(* IEC 61131-3 sources: Std_PalletMover/Class/Curtis_Base, 1 file *)

(* ---- Curtis_Base.st ---- *)
//#Define cNoNmtIfOk
#Define cCommTo                   1000    // 1000
#Define cHeartBeat                150     // 1000 Every 1 Sec.
#define COMM_TIMEOUT              1000    // ms before timeout
#define PDO1_SEND_INTERVAL        40      // 100 ms
#define TIMEOUTDELAY              15000    // Delay before checking for a communication timeout.
#define REFERENCETIMEOUT          30 SEC  //
#define FUSE_BAD_TIME             4 SEC
#define MAX_TIME_DRIVE_MODE_REQ   150 //ms

(*!
<Class
	Name               = "Curtis_Base"
	Revision           = "0.0"
	RealtimeTask       = "false"
	CyclicTask         = "false"
	DefCyclictime      = "5 ms"
	BackgroundTask     = "false"
	Sigmatek           = "false"
	OSInterface        = "false"
	HighPriority       = "false"
	Automatic          = "false"
	UpdateMode         = "Prescan"
	IconPath           = ".\Class\Curtis_1232E_FR\curtis.ico"
	SharedCommandTable = "true"
	Objectsize         = "(510,300)"
	Comment            = "CAN Message for Curtis Drives">
	<Channels>
		<Server Name="Active" Visualized="true" Initialize="false" WriteProtected="true" Retentive="false"/>
		<Server Name="AI_BrakePot" Visualized="true" Initialize="false" WriteProtected="true" Retentive="false"/>
		<Server Name="AI_ThrottlePot" Visualized="true" Initialize="false" WriteProtected="true" Retentive="false"/>
		<Server Name="AutoAccelTime" Visualized="true" Initialize="true" DefValue="100" WriteProtected="false" Retentive="SRam" Comment="0,1 second acceleration time"/>
		<Server Name="AutoAct" Visualized="true" Initialize="false" WriteProtected="true" Retentive="false"/>
		<Server Name="AutoDecelTime" Visualized="true" Initialize="true" DefValue="10" WriteProtected="false" Retentive="SRam" Comment="0,1 second acceleration time"/>
		<Server Name="AutomaticSetpoint" Visualized="true" Initialize="false" WriteProtected="false" Retentive="false"/>
		<Server Name="AutoSetp" Visualized="true" Initialize="false" WriteProtected="true" Retentive="false"/>
		<Server Name="BDI" Visualized="true" Initialize="false" WriteProtected="true" Retentive="false"/>
		<Server Name="BrakePotSigned" Visualized="true" Initialize="true" WriteProtected="false" Retentive="File"/>
		<Server Name="Capacitor_Voltage" Visualized="true" Initialize="false" WriteProtected="true" Retentive="false"/>
		<Server Name="ClassSvr" Visualized="false" Initialize="false" WriteProtected="true" Retentive="false"/>
		<Server Name="CommunicationOk" Visualized="true" Initialize="false" WriteProtected="true" Retentive="false"/>
		<Server Name="DriveMode" Visualized="true" Initialize="false" WriteProtected="true" Retentive="false"/>
		<Server Name="DriveModeRequest" Visualized="true" Initialize="false" WriteProtected="false" Retentive="false"/>
		<Server Name="EmStopOk" Visualized="true" Initialize="false" WriteProtected="true" Retentive="false"/>
		<Server Name="Enabled" Visualized="true" Initialize="true" DefValue="1" WriteProtected="false" Retentive="File"/>
		<Server Name="I_DigitalOut6" Visualized="true" Initialize="false" WriteProtected="true" Retentive="false" Comment="Sw_14"/>
		<Server Name="I_DigitalOut7" Visualized="true" Initialize="false" WriteProtected="true" Retentive="false" Comment="Sw_15"/>
		<Server Name="I_Driver1" Visualized="true" Initialize="false" WriteProtected="true" Retentive="false" Comment="Sw_9&#13;&#10;Auger_1 - bI_SP_HighLow"/>
		<Server Name="I_Driver2" Visualized="true" Initialize="false" WriteProtected="true" Retentive="false" Comment="Sw_10&#13;&#10;Auger_1 - bI_AugerOnOff"/>
		<Server Name="I_Driver3" Visualized="true" Initialize="false" WriteProtected="true" Retentive="false" Comment="Sw_11&#13;&#10;Auger_1 - bSP_HighLow"/>
		<Server Name="I_Driver4" Visualized="true" Initialize="false" WriteProtected="true" Retentive="false" Comment="Sw_12&#13;&#10;Auger_1 - bAugerOnOff"/>
		<Server Name="I_PropDriver" Visualized="true" Initialize="false" WriteProtected="true" Retentive="false" Comment="Sw_13&#13;&#10;Pin 2"/>
		<Server Name="I_Switch1" Visualized="true" Initialize="false" WriteProtected="true" Retentive="false" Comment="Pin 24 - Switch 1"/>
		<Server Name="I_Switch16" Visualized="true" Initialize="false" WriteProtected="true" Retentive="false" Comment="Pin 14 - Switch 16"/>
		<Server Name="I_Switch2" Visualized="true" Initialize="false" WriteProtected="true" Retentive="false" Comment="Pin 8 - Switch 2"/>
		<Server Name="I_Switch3" Visualized="true" Initialize="false" WriteProtected="true" Retentive="false" Comment="Pin 9 - Switch 3"/>
		<Server Name="I_Switch4" Visualized="true" Initialize="false" WriteProtected="true" Retentive="false" Comment="Pin 10 - Switch 4"/>
		<Server Name="I_Switch5" Visualized="true" Initialize="false" WriteProtected="true" Retentive="false" Comment="Pin 11 - Switch 5"/>
		<Server Name="I_Switch6" Visualized="true" Initialize="false" WriteProtected="true" Retentive="false" Comment="Pin 12 - Switch 6"/>
		<Server Name="I_Switch7" Visualized="true" Initialize="false" WriteProtected="true" Retentive="false" Comment="Pin 22 - Switch 7"/>
		<Server Name="I_Switch8" Visualized="true" Initialize="false" WriteProtected="true" Retentive="false" Comment="Pin 33 - Switch 8"/>
		<Server Name="InterlockExternal1" Visualized="true" Initialize="false" WriteProtected="true" Retentive="false"/>
		<Server Name="InterlockExternal2" Visualized="true" Initialize="false" WriteProtected="true" Retentive="false"/>
		<Server Name="InterlockFeedback" Visualized="true" Initialize="false" WriteProtected="true" Retentive="false"/>
		<Server Name="MotorCurrent" Visualized="true" Initialize="false" WriteProtected="true" Retentive="false"/>
		<Server Name="MotorRPM" Visualized="true" Initialize="false" WriteProtected="true" Retentive="false" Comment="Speed of Motor"/>
		<Server Name="MotorTemperature" Visualized="true" Initialize="false" WriteProtected="true" Retentive="false"/>
		<Server Name="QD_DigitalOut6" Visualized="true" Initialize="false" WriteProtected="false" Retentive="false" Comment="Auger_1 - Horn"/>
		<Server Name="QD_DigitalOut7" Visualized="true" Initialize="false" WriteProtected="false" Retentive="false" Comment="Auger_1 - bDrive_OnOff"/>
		<Server Name="QD_Driver1" Visualized="true" Initialize="false" WriteProtected="false" Retentive="false" Comment="Auger_1 - Pin 6 - bQ_Actu_L_In"/>
		<Server Name="QD_Driver2" Visualized="true" Initialize="false" WriteProtected="false" Retentive="false" Comment="Auger_1 - Pin 5 - bQ_Actu_L_Out"/>
		<Server Name="QD_Driver3" Visualized="true" Initialize="false" WriteProtected="false" Retentive="false" Comment="Auger_1 - Pin 4 - bQ_Actu_R_In"/>
		<Server Name="QD_Driver4" Visualized="true" Initialize="false" WriteProtected="false" Retentive="false" Comment="Auger_1 - Pin 3 - bQ_Actu_R_Out"/>
		<Server Name="QD_PropDriver" Visualized="true" Initialize="false" WriteProtected="false" Retentive="false"/>
		<Server Name="Referenced" Visualized="true" Initialize="false" WriteProtected="true" Retentive="false"/>
		<Server Name="ThrottlePotSigned" Visualized="true" Initialize="true" WriteProtected="false" Retentive="File"/>
		<Client Name="_CanOpenBaseRiwo" Required="true" Internal="true"/>
		<Client Name="AlarmStartId" Required="true" Internal="false"/>
		<Client Name="NodeId" Required="true" Internal="false"/>
		<Client Name="objDriver" Required="false" Internal="false"/>
	</Channels>
	<Separators>
		<Servers>
			<SepChn Position="34"/>
			<SepChn Position="38"/>
		</Servers>
	</Separators>
	<RevDoku>
		<Owner Company="RIWO Engineering BV" Author="P vd Voort"/>
		<Dokumentation Revision="0.0" Date="2022-08-29" Author="P vd Voort" Company="RIWO Engineering BV" Description="First Build Up"/>
	</RevDoku>
	<Network Name="Curtis_Base">
		<!-- List of Components in this network -->
		<Components>
			<Object
				Name       = "_CanOpenBaseRiwo"
				Class      = "CanOpenBaseRiwo"
				Position   = "(390,240)"
				Visualized = "true"
				CyclicTime = "1 ms">
				<Channels>
					<Server Name="Server0"/>
					<Client Name="cNode" Value="1"/>
					<Client Name="ConfigData"/>
					<Client Name="Driver"/>
				</Channels>
			</Object>
		</Components>
		<Comments>
		</Comments>
		<!-- List of Connections in this network -->
		<Connections>
			<Connection Source="this._CanOpenBaseRiwo" Destination="_CanOpenBaseRiwo.Server0"/>
			<Connection Source="_CanOpenBaseRiwo.Driver" Destination="this.objDriver" Vertices="(390,330),(38,330),"/>
			<Connection Source="_CanOpenBaseRiwo.cNode" Destination="this.NodeId" Vertices="(390,390),(38,270),"/>
		</Connections>
		<!-- Headerfiles -->
		<Options>
		</Options>
	</Network>
</Class>
*)
Curtis_Base : CLASS
	TYPE
#pragma pack(push, 1)
	  CurtisMessageConfig : STRUCT
	    Byte0 : BSINT
	    [
	      1 Q1,
	      2 Q1not,
	      3 Q2,
	      4 Q2not,
	      5 Bit4,
	      6 Bit5,
	      7 Bit6,
	      8 Bit7,
	    ];
	    Byte1 : BSINT
	    [
	      1 InputState_A,
	      2 InputState_B,
	      3 InputState_C,
	      4 InputState_D,
	      5 Bit4,
	      6 Bit5,
	      7 Bit6,
	      8 InputState_StandBy,
	    ];
	    Byte2 : BSINT
	    [
	      1 Bit0_SwFldQ1,
	      2 Bit1_SwFldQ1,
	      3 Bit2_SwFldQ1,
	      4 Bit3_SwFldQ1,
	      5 Bit4_SwFldQ1,
	      6 Bit5,
	      7 Bit6,
	      8 Bit7,
	    ];
	    Byte3 : BSINT
	    [
	      1 Bit0_SwFldQ2,
	      2 Bit1_SwFldQ2,
	      3 Bit2_SwFldQ2,
	      4 Bit3_SwFldQ2,
	      5 Bit4_SwFldQ2,
	      6 Bit5,
	      7 Bit6,
	      8 Bit7,
	    ];
	    Byte4 : BSINT
	    [
	      1 Bit0_DeviceStatus,
	      2 Bit1_DeviceStatus,
	      3 Bit2_DeviceStatus,
	      4 Bit3_DeviceStatus,
	      5 Bit4,
	      6 Bit5,
	      7 Bit6,
	      8 Bit7,
	    ];
	    Byte5 : SINT;
	    Byte6and7 : INT;
	  END_STRUCT;
#pragma pack(pop)
	  CurtisSendConfig : BSINT
	  [
	    1 VirtInp_A,
	    2 VirtInp_B,
	    3 VirtInp_C,
	    4 VirtInp_D,
	    5 Bit4,
	    6 Bit5,
	    7 Bit6,
	    8 VirtInp_Standby,
	  ];
	  eCurtisAlarms :
	  (
	    ca_MainContactor_Welded:=1,
	    ca_MainContactor_NotClosed:=2,
	    ca_PotLow:=3,
	    ca_ThrottleLow:=4,
	    ca_ThrottleHigh:=5,
	    ca_Pot2Low:=6,
	    ca_Pot2High:=7,
	    ca_EepromFail:=8,
	    ca_SequenceFault:=9,
	    ca_UnderVoltage:=10,
	    ca_OverVoltage:=11,
	    ca_UnderVoltage_CutBack:=12,
	    ca_OverVoltage_CutBack:=13,
	    ca_FuseBad:=14,
	    ca_ControllerTemp_CutBack:=15,
	    ca_Controller_UnderTemp:=16,
	    ca_Controller_OverTemp:=17,
	    ca_Coil1_Short:=18,
	    ca_Coil2_Short:=19,
	    ca_Coil3_Short:=20,
	    ca_Coil4_Short:=21,
	    ca_PD_Short:=22,
	    ca_Main_Short:=23,
	    ca_EmBrake_Short:=24,
	    ca_PreCharge_Failed:=25,
	    ca_Digital6_OverCurrent:=26,
	    ca_Digital7_OverCurrent:=27,
	    ca_Controller_OverCurrent:=28,
	    ca_CurrentSensor_Fault:=29,
	    ca_MotorTemp_CutBack:=30,
	    ca_ParameterChange_Fault:=31,
	    ca_Motor_Open:=32,
	    ca_ExtSupply_OutofRange:=33,
	    ca_MotorTemp_SensorFault:=34,
	    ca_VC1_RunTime:=35,
	    ca_5vSupply_Failure:=36,
	    ca_OSGeneral:=37,
	    ca_PDO_Timeout:=38,
	    ca_Encoder_Fault:=39,
	    ca_StallDetected:=40,
	    ca_Com_Timeout:=41,
	    ca_NotRef:=42,
	    ca_RevHpd:=43,
	    ca_NotEnabled:=44,
	    ca_MotorType_Fault:=45,
	    ca_SuperVision:=46,
	    ca_MotorCharacter:=47,
	    ca_PumpHardware:=48,
	    ca_NotDefined_1:=49,
	    ca_VCL_Mismatch:=50,
	    ca_EmBrake_Failed:=51,
	    ca_Encoder_Lose:=52,
	    ca_Rev_Timeout:=53,
	    ca_Dual_Fault:=54,
	    ca_TractionController_Fault:=55,
	    ca_Illegal_ModelNumber:=56,
	    ca_PumpOverCurrent:=57,
	    ca_PumpBdi:=58,
	    ca_PumpHpd:=59,
	    ca_DualMotor_Par_MisMatch:=60,
	    ca_NotDefined_2:=61,
	    ca_NotDefined_3:=62,
	    ca_NotDefined_4:=63,
	    ca_EncoderPulse:=64
	  )$UDINT;
	  eCurtisDriveMode :  //! <Type Public="true" Name="eCurtisDriveMode"/>
	  (
	    cdm_Idle,
	    cdm_TimeOut,
	    cdm_EmergencyStop,
	    cdm_Referencing,
	    cdm_Manual,
	    cdm_Auto,
	    cdm_DriveReset,
	    cdm_ExtInterlockReset
	  )$UDINT;
	  eCurtisDriveModeRequest :  //! <Type Public="true" Name="eCurtisDriveModeRequest"/>
	  (
	    cdmr_NoReq:=4294967295,
	    cdmr_Idle,
	    cdmr_Reference,
	    cdmr_Manual:=2,
	    cdmr_Automatic:=3,
	    cdmr_ResetDrive:=4,
	    cdmr_ResetExtInterlock:=5
	  )$DINT;
#pragma pack(push, 1)
	  Errors : STRUCT
	    Error1 : DINT;
	    Error2 : DINT;
	    Error3 : DINT;
	    Error4 : DINT;
	    Error5 : DINT;
	    Error6 : DINT;
	    Error7 : DINT;
	    NumberOfErrors : DINT;
	  END_STRUCT;
#pragma pack(pop)
	  FuncComm :
	  (
	    _StandBy,
	    _Read,
	    _Write,
	    _Busy
	  )$UDINT;
#pragma pack(push, 1)
	  PdoSplit : STRUCT
	    Val1 : HSINT;
	    Val2 : HSINT;
	    Val3 : HSINT;
	    Val4 : HSINT;
	    Val5 : HSINT;
	    Val6 : HSINT;
	    Val7 : HSINT;
	    Val8 : HSINT;
	  END_STRUCT;
#pragma pack(pop)
	END_TYPE
  //Servers:
	ClassSvr 	: SvrChCmd_DINT;
	Active 	: SvrCh_DINT;
	CommunicationOk 	: SvrCh_DINT;
	DriveMode 	: SvrCh_eCurtisDriveMode_PTofCls_Curtis_Base;
	EmStopOk 	: SvrCh_DINT;
	Referenced 	: SvrCh_DINT;
	InterlockFeedback 	: SvrCh_DINT;
	InterlockExternal1 	: SvrCh_DINT;
	InterlockExternal2 	: SvrCh_DINT;
	AutoAct 	: SvrCh_DINT;
	AutoSetp 	: SvrCh_DINT;
	MotorCurrent 	: SvrCh_DINT;
	BDI 	: SvrCh_DINT;
	Capacitor_Voltage 	: SvrCh_DINT;
	MotorTemperature 	: SvrCh_DINT;
	AI_ThrottlePot 	: SvrCh_DINT;
	AI_BrakePot 	: SvrCh_DINT;
	I_Switch1 	: SvrCh_DINT;
	I_Switch2 	: SvrCh_DINT;
	I_Switch3 	: SvrCh_DINT;
	I_Switch4 	: SvrCh_DINT;
	I_Switch5 	: SvrCh_DINT;
	I_Switch6 	: SvrCh_DINT;
	I_Switch7 	: SvrCh_DINT;
	I_Switch8 	: SvrCh_DINT;
	I_Driver1 	: SvrCh_DINT;
	I_Driver2 	: SvrCh_DINT;
	I_Driver3 	: SvrCh_DINT;
	I_Driver4 	: SvrCh_DINT;
	I_PropDriver 	: SvrCh_DINT;
	I_DigitalOut6 	: SvrCh_DINT;
	I_DigitalOut7 	: SvrCh_DINT;
	I_Switch16 	: SvrCh_DINT;
	MotorRPM 	: SvrCh_DINT;
	Enabled 	: SvrCh_DINT;
	ThrottlePotSigned 	: SvrCh_DINT;
	BrakePotSigned 	: SvrCh_DINT;
	DriveModeRequest 	: SvrCh_eCurtisDriveModeRequest_PTofCls_Curtis_Base;
	AutomaticSetpoint 	: SvrCh_DINT;
	AutoAccelTime 	: SvrCh_DINT;
	AutoDecelTime 	: SvrCh_DINT;
	QD_Driver1 	: SvrCh_DINT;
	QD_Driver2 	: SvrCh_DINT;
	QD_Driver3 	: SvrCh_DINT;
	QD_Driver4 	: SvrCh_DINT;
	QD_PropDriver 	: SvrCh_DINT;
	QD_DigitalOut6 	: SvrCh_DINT;
	QD_DigitalOut7 	: SvrCh_DINT;
  //Clients:
	AlarmStartId 	: CltCh_DINT;
	NodeId 	: CltCh_DINT;
	objDriver 	: CltChCmd_CanDriverBase;
	_CanOpenBaseRiwo 	: CltChCmd_CanOpenBaseRiwo;
  //Variables:
		_pdoIn1 	: PDOStr;
		_pdo1rxTime 	: UDINT;
		_pdoIn2 	: PDOStr;
		_pdo2rxTime 	: UDINT;
		_pdoIn3 	: PDOStr;
		_pdo3rxTime 	: UDINT;
		_pdoIn4 	: PDOStr;
		_pdo4rxTime 	: UDINT;
		_pdo1Out 	: PDOStr;
		_initCntr 	: DINT;
		_prevReferenced 	: DINT;
		_notReferencedStartTime 	: UDINT;
		_sendPDO1TimeStamp 	: UDINT;
		_sendPDO2TimeStamp 	: UDINT;
		_timeoutDelayStart 	: UDINT;
		_StartupDelayActive 	: BOOL;
		_tempOk 	: BOOL;
		_DriveCycleTimeOk 	: BOOL;
		_pdo1RxInterval 	: UDINT;
		_FuseBadStartTime 	: UDINT;
		_DriveModeReqStepper 	: DINT;
		_IntDriveModeReq 	: eCurtisDriveModeRequest;
		_DriveModeRequestTime 	: UDINT;
		_pObjCurtis_Universal 	: ^Curtis_Universal;
  //Functions:

	FUNCTION VIRTUAL GLOBAL Init;

	FUNCTION VIRTUAL _split16bit
		VAR_INPUT
			Input16bit 	: INT;
			pLSB 	: ^HSINT;
			pMSB 	: ^HSINT;
		END_VAR;

	FUNCTION VIRTUAL _receiveData;

	FUNCTION VIRTUAL _to16bit
		VAR_INPUT
			LSB 	: HSINT;
			MSB 	: HSINT;
		END_VAR
		VAR_OUTPUT
			Output16bit 	: UINT;
		END_VAR;

	FUNCTION VIRTUAL _sendData;

	FUNCTION VIRTUAL _handleDriveMode;

	FUNCTION GLOBAL GetThis
		VAR_OUTPUT
			pObject 	: ^void;
		END_VAR;

	FUNCTION GLOBAL SetObjCurtis_Universal
		VAR_INPUT
			pObject 	: ^void;
		END_VAR;
  //Tables:
	FUNCTION @STD
		VAR_OUTPUT
			ret_code	: CONFSTATES;
		END_VAR;
	FUNCTION GLOBAL TAB @CT_;
END_CLASS;

#pragma using CanOpenBaseRiwo
#pragma usingLtd CanDriverBase

#pragma usingLtd Curtis_Universal

(*****************************************************************************************
	Curtis Motor Controller CAN-OPEN driver
	****************************************************************************************
  This class cummunicates with a Curtis 1232 Motor Controller over CAN-OPEN.
  - write RPM and outputs to the Encoder and receive inputs
	****************************************************************************************
*)
FUNCTION VIRTUAL GLOBAL Curtis_Base::Init

  _initCntr += 1;

  case _initCntr of
   1:

    2:
    //** Larger than 10, get info from external classes is enabled **\\
    12:
      _timeoutDelayStart := ops.tAbsolute;
      _StartupDelayActive := TRUE;
  end_case;

END_FUNCTION

FUNCTION VIRTUAL Curtis_Base::_handleDriveMode

END_FUNCTION

FUNCTION VIRTUAL Curtis_Base::_receiveData
  //overide

END_FUNCTION

FUNCTION VIRTUAL Curtis_Base::_sendData

END_FUNCTION
(*****************************************************************************************************)
(** _handleAlarmStates
(** function handles every specific alarm reset if allowed the allarm is set inactive
(*****************************************************************************************************)
FUNCTION VIRTUAL Curtis_Base::_split16bit
	VAR_INPUT
		Input16bit 	: INT;
		pLSB 	: ^HSINT;
		pMSB 	: ^HSINT;
	END_VAR

    pLSB^ := (Input16bit and 16#00FF)$hsint;
    pMSB^ := ((Input16bit and 16#FF00)shr 8)$hsint;

END_FUNCTION

FUNCTION VIRTUAL Curtis_Base::_to16bit
	VAR_INPUT
		LSB 	: HSINT;
		MSB 	: HSINT;
	END_VAR
	VAR_OUTPUT
		Output16bit 	: UINT;
	END_VAR

  Output16bit := (MSB shl 8) or LSB;

END_FUNCTION

FUNCTION GLOBAL Curtis_Base::GetThis
	VAR_OUTPUT
		pObject 	: ^void;
	END_VAR

  pObject := this ;

END_FUNCTION

FUNCTION GLOBAL Curtis_Base::SetObjCurtis_Universal
	VAR_INPUT
		pObject 	: ^void;
	END_VAR

  _pObjCurtis_Universal:= pObject$^Curtis_Universal ;

END_FUNCTION
